FUNCTION_BLOCK KinematicGroup_TcEvents EXTENDS CyclicComponent IMPLEMENTS I_EventReactionTcEvents
VAR
	KinematicGroup : I_KinematicGroup;
	Events		   : TcEventClass('Kinematic Group Events');
END_VAR

METHOD CyclicLogic
IF KinematicGroup = 0 THEN
	RETURN;
END_IF

IF KinematicGroup.Error THEN
	Events.Arguments(E_KinematicGroup.KinematicGroupError).Clear().AddString(TO_STRING(KinematicGroup.ErrorId));
	Events.RaiseEvent(E_KinematicGroup.KinematicGroupError);
END_IF
END_METHOD

(*FB_Init is always available implicitly and it is used primarily for initialization.
The return value is not evaluated. For a specific influence, you can also declare the
methods explicitly and provide additional code there with the standard initialization
code. You can evaluate the return value.*)
METHOD FB_Init : BOOL
VAR_INPUT
	(* TRUE: the retain variables are initialized (reset warm / reset cold)*)
	bInitRetains : BOOL;

	(* TRUE: the instance will be copied to the copy code afterward (online change)   *)
	bInCopyCode	   : BOOL;
	Name		   : T_MaxString;
	KinematicGroup : I_KinematicGroup;
END_VAR
THIS^.KinematicGroup := KinematicGroup;
Events.GenerateTcEvents(KinematicGroup.Name, ADR(TC_Events.KinematicGroup), SIZEOF(ST_KinematicGroup));
END_METHOD

METHOD GetHighestActiveEventReaction : DINT
GetHighestActiveEventReaction := Events.GetHighestActiveEventReaction();
END_METHOD

METHOD GetHighestActiveEventSeverity : TcEventSeverity
GetHighestActiveEventSeverity := Events.GetHighestActiveEventSeverity();
END_METHOD

METHOD Reset
Events.Reset();
END_METHOD

METHOD SetEventReactions
VAR_INPUT
	Verbose	 : DINT := 0;
	Info	 : DINT := 1;
	Warning	 : DINT := 2;
	Error	 : DINT := 3;
	Critical : DINT := 4;
END_VAR
Events.SetEventReactions(Verbose,
						 Info,
						 Warning,
						 Error,
						 Critical);
END_METHOD

END_FUNCTION_BLOCK

(* stored: Version 1.1.0.1, ProductVersion 3.1.4026.18
   POU KinematicGroup_TcEvents: Id {21b161f7-eb7b-49f9-8d98-88b558d342ec}, SpecialFunc None
   Folder Events: Id {331363c2-64fb-4d3d-b501-2891e295f8b3}
   Method CyclicLogic: Id {eb8680de-c9e2-4b02-a42a-cca529595784}
   Method FB_Init: Id {8c63b2d9-3f3a-49d8-8731-91accf010af6}
   Method GetHighestActiveEventReaction: Id {771d3874-e818-4177-ab63-55e69664e46a}
   Method GetHighestActiveEventSeverity: Id {697476d1-0abf-4051-b201-fe87218471ff}
   Method Reset: Id {717622c2-e543-40e8-9070-11913164f5b7}
   Method SetEventReactions: Id {b490104d-3824-4f2d-b581-58a0275d0d0a} *)
